FUNCTION F_DeviceTwin_GetSubscriberTopicStatusCodes : STRING
VAR_INPUT
END_VAR
VAR
END_VAR

F_DeviceTwin_GetSubscriberTopicStatusCodes := '$$iothub/twin/res/#';

END_FUNCTION

(* stored: Version 1.1.0.1, ProductVersion 3.1.4022.3
   POU F_DeviceTwin_GetSubscriberTopicStatusCodes: Id {a932b92c-041d-4788-a4a7-741c8e5b30ac}, SpecialFunc None *)
